(* IEC 61131-3 sources: plc-home-automation/home_automation/lighting_heating_updated/src/utils/io, 6 files *)

(* ---- AfterBurnerOutput.st ---- *)
FUNCTION_BLOCK AfterBurnerOutput
  VAR_INPUT CONSTANT
    name : STRING;
  END_VAR

  VAR_INPUT
    delay : TIME;
    duration: TIME;
    feedOn: BOOL R_EDGE;
    feedOff : BOOL R_EDGE;
    emergencyStop : BOOL R_EDGE;
  END_VAR

  VAR_OUTPUT
    out: BOOL := FALSE;
  END_VAR

  VAR
    delayTimer: TON;
    delayTimerInput: BOOL;
    durationTimer: TON;
    durationTimerInput: BOOL;
    sentence : STRING;
  END_VAR

  IF feedOn THEN
     delayTimerInput := TRUE;
     sentence := CONCAT(name, ' started ramping up');
     SWITCH_TRACKER(name := sentence);
  END_IF;

  IF feedOff THEN
     delayTimerInput := FALSE;
     sentence := CONCAT(name, ' stopped ramping up');
     SWITCH_TRACKER(name := sentence);
  END_IF;

  delayTimer(IN := delayTimerInput, PT := delay);

  IF delayTimer.Q THEN
     durationTimer(IN := FALSE, PT := duration); // Reset ongoing output cycle
     durationTimerInput := TRUE;
     out := TRUE;
     delayTimerInput := FALSE;
     sentence := CONCAT(name, ' turned on and resetted previous cycle');
     SWITCH_TRACKER(name := sentence);
  END_IF;

  durationTimer(IN := durationTimerInput, PT := duration);

  IF durationTimer.Q THEN
     durationTimerInput := FALSE;
     out := FALSE;
     sentence := CONCAT(name, ' turned off');
     SWITCH_TRACKER(name := sentence);
  END_IF;

  IF emergencyStop THEN
     out := FALSE;
     delayTimerInput := FALSE;
     durationTimerInput := FALSE;
  END_IF;
END_FUNCTION_BLOCK // AfterBurnerOutput

(* ---- ChangeOnOff.st ---- *)
FUNCTION_BLOCK ChangeOnOff
  VAR_INPUT CONSTANT
    name : STRING;
  END_VAR

  VAR_INPUT
    requestOn : BOOL R_EDGE;
    requestOff: BOOL R_EDGE;
    requestChange : BOOL R_EDGE;
  END_VAR

  VAR_OUTPUT
    output: BOOL := FALSE;
  END_VAR

  VAR
     sentence : STRING;
  END_VAR

    IF (requestOn AND NOT requestOff AND NOT requestChange) THEN
      sentence := CONCAT(name, ' on');
      SWITCH_TRACKER(name := sentence);
      output := TRUE;
    ELSIF (NOT requestOn AND requestOff AND NOT requestChange) THEN
      sentence := CONCAT(name, ' off');
      SWITCH_TRACKER(name := sentence);
      output := FALSE;
    ELSIF (NOT requestOn AND NOT requestOff AND requestChange) THEN
      sentence := CONCAT(name, ' changed');
      SWITCH_TRACKER(name := sentence);
      output := NOT output;
    END_IF;

END_FUNCTION_BLOCK

(* ---- DurationOut.st ---- *)
FUNCTION_BLOCK InterruptableReentrantDurationOut
  VAR_INPUT
     onSignal : BOOL R_EDGE;
     offSignal : BOOL R_EDGE;
     duration : time;
     name : STRING;
  END_VAR

  VAR_OUTPUT
     active : BOOL;
  END_VAR

  VAR
     timer : TON;
     timerTrigger: BOOL := false;
     sentence : STRING;
  END_VAR

  IF onSignal THEN
     timerTrigger := true;
     timer(IN := false, PT := duration);
     active := true;
     sentence := CONCAT(name, ' on');
     SWITCH_TRACKER(name := sentence);
  END_IF;

  IF offSignal THEN
     timerTrigger := false;
     timer(IN := false, PT := duration);
     active := false;
     sentence := CONCAT(name, ' interrupted');
     SWITCH_TRACKER(name := sentence);
  END_IF;

  IF timer.Q THEN
     timerTrigger := false;
     active := false;
     sentence := CONCAT(name, ' off');
     SWITCH_TRACKER(name := sentence);
  END_IF;

  timer(IN := timerTrigger, PT := duration);
END_FUNCTION_BLOCK

FUNCTION_BLOCK ReentrantDurationOut
  VAR_INPUT
     onSignal : BOOL R_EDGE;
     duration : time;
     name : STRING;
  END_VAR

  VAR_OUTPUT
     active : BOOL;
  END_VAR

  VAR
     timer : TON;
     timerTrigger: BOOL := false;
     sentence: STRING;
  END_VAR

  IF onSignal THEN
     timerTrigger := true;
     timer(IN := false, PT := duration);
     active := true;
     sentence := CONCAT(name, ' on');
     SWITCH_TRACKER(name := sentence);
  END_IF;

  IF timer.Q THEN
     timerTrigger := false;
     active := false;
     sentence := CONCAT(name, ' off');
     SWITCH_TRACKER(name := sentence);
  END_IF;

  timer(IN := timerTrigger, PT := duration);
END_FUNCTION_BLOCK

FUNCTION_BLOCK DurationOut
  VAR_INPUT
     onSignal : BOOL R_EDGE;
     duration : time;
     name: STRING;
  END_VAR

  VAR_OUTPUT
     active : BOOL;
  END_VAR

  VAR
     timer : TON;
     timerTrigger: BOOL := false;
     sentence: STRING;
  END_VAR

  IF onSignal THEN
     timerTrigger := true;
     active := true;
     sentence := CONCAT(name, ' on');
     SWITCH_TRACKER(name := sentence);
  END_IF;

  IF timer.Q THEN
     timerTrigger := false;
     active := false;
     sentence := CONCAT(name, ' off');
     SWITCH_TRACKER(name := sentence);
  END_IF;

  timer(IN := timerTrigger, PT := duration);
END_FUNCTION_BLOCK

(* ---- InPlaceOnOff.st ---- *)
FUNCTION_BLOCK InPlaceOnOff
    VAR_INPUT
      onSignal : BOOL R_EDGE;
      offSignal : BOOL R_EDGE;
    END_VAR
    VAR_IN_OUT
      name: STRING;
      controlledVariable : BOOL;
    END_VAR

    VAR
      sentence : STRING;
    END_VAR

    IF onSignal THEN
       controlledVariable := TRUE;
       sentence := CONCAT(name, ' is ON');
       SWITCH_TRACKER(name := sentence);
    END_IF;
    IF offSignal THEN
       controlledVariable := FALSE;
       sentence := CONCAT(name, ' is OFF');
       SWITCH_TRACKER(name := sentence);
    END_IF;
END_FUNCTION_BLOCK

(* ---- OnThenOffPulse.st ---- *)
FUNCTION_BLOCK OnThenOffPulse
  VAR_INPUT
     timeOn   : TIME;
     timeOff  : TIME;
     onSignal : BOOL R_EDGE;
  END_VAR

  VAR_OUTPUT
     active : BOOL;
  END_VAR

  VAR
     out : DurationOut;
     idle: DurationOut;
     outTrigger : BOOL := false;
     idleTrigger :  BOOL := false;
  END_VAR

  IF NOT out.active AND outTrigger THEN
     outTrigger := false;
     idleTrigger := true;
     active := false;
  END_IF;

  IF onSignal AND ( NOT (idle.active OR out.active) ) THEN
     outTrigger := true;
     idleTrigger := false;
     active := true;
  END_IF;

  out(onSignal := outTrigger, duration := timeOn);
  idle(onSignal := idleTrigger, duration := timeOff);
END_FUNCTION_BLOCK

(* ---- RoomSwitch.st ---- *)
FUNCTION_BLOCK RoomSwitch
(*API for normally open room push switches.*)
    VAR_INPUT
      onSignal : BOOL R_EDGE;
    END_VAR
    VAR_IN_OUT
      name: STRING;
    END_VAR
    VAR_OUTPUT
      out : BOOL := FALSE;
    END_VAR

    IF onSignal THEN
       out := NOT out;
       SWITCH_TRACKER(name := name);
    END_IF;
END_FUNCTION_BLOCK
